{attribute addProperty BoxType "EL6080-0000-0018"}
{attribute addProperty Id "StatusAT %I*Status_8B1CA2AE1620InputsEMPTY_STRUCTURE000ControlAT %Q*Control_734938A41620OutputsEMPTY_STRUCTURE000WcStateAT %I*WcState_F855686C1620InfoDataAT %I*InfoData_BC63D37F80100"}
{attribute addProperty CRC "2111624504"}
{attribute addProperty SizeInBites "128"}
{attribute addProperty SizeInBytes "16"}
TYPE EL6080_820BDBFD :
STRUCT
	{attribute addProperty Name "Status"}
	Status : Status_8B1CA2AE;
	{attribute addProperty Name "Inputs"}
	Inputs : EMPTY_STRUCTURE;
	{attribute addProperty Name "Control"}
	Control : Control_734938A4;
	{attribute addProperty Name "Outputs"}
	Outputs : EMPTY_STRUCTURE;
	{attribute addProperty Name "WcState"}
	WcState : WcState_F855686C;
	{attribute addProperty Name "InfoData"}
	InfoData : InfoData_BC63D37F;
END_STRUCT
END_TYPE

(* stored: Version 1.2.0.0, ProductVersion 3.1.4024.9
   DUT EL6080_820BDBFD: Id {7b56521b-4870-456e-8ee6-1ed1ae228b10} *)
